SUBAPPLICATION Uebung_035a1_AX (* Ampelsteuerung mit Pattern Sequencer (AX) *)
  (* Standard: 61499-2; Description: Copyright (c) 2023 Meisterschulen am Ostbahnhof This program and the accompanying materials are made available under the terms of the Eclipse Public License 2.0 which is available at https://www.eclipse.org/legal/epl-2.0/ SPDX-License-Identifier: EPL-2.0 *)
  (* Version 1.0, 2026-02-01, Franz Höpfinger, Meisterschulen am Ostbahnhof, initial API and implementation and/or initial documentation *)
  PACKAGE Uebungen;
  IMPORT logiBUS::io::DI::logiBUS_DI::Input_I1;
  IMPORT logiBUS::io::DI::logiBUS_DI_Events::BUTTON_SINGLE_CLICK;
  IMPORT logiBUS::io::DQ::logiBUS_DO::Output_Q1;
  IMPORT logiBUS::io::DQ::logiBUS_DO::Output_Q2;
  IMPORT logiBUS::io::DQ::logiBUS_DO::Output_Q3;
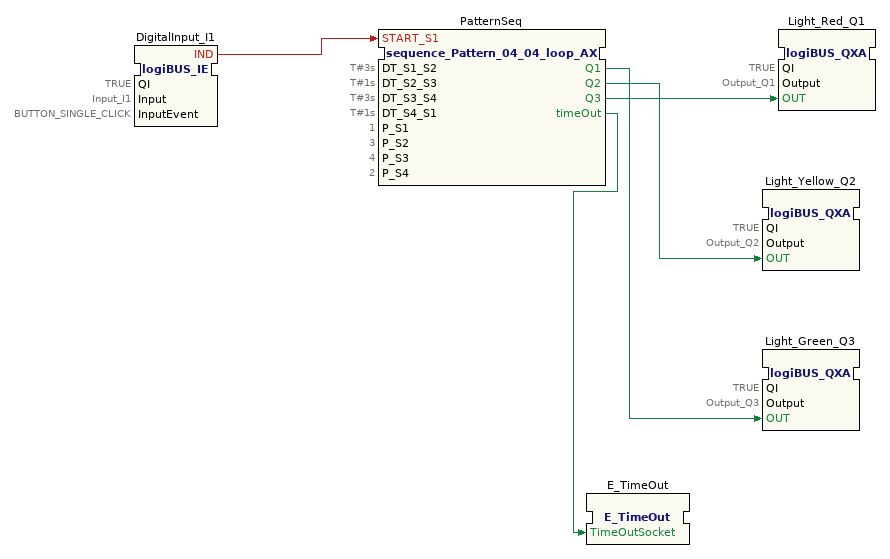
  FBS
    PatternSeq : logiBUS::utils::sequence::pattern::sequence_Pattern_04_04_loop_AX(DT_S1_S2 := T#3s, DT_S2_S3 := T#1s, DT_S3_S4 := T#3s, DT_S4_S1 := T#1s, P_S1 := 1, P_S2 := 3, P_S3 := 4, P_S4 := 2);
    DigitalInput_I1 : logiBUS::io::DI::logiBUS_IE(QI := TRUE, Input := Input_I1, InputEvent := BUTTON_SINGLE_CLICK);
    Light_Red_Q1 : logiBUS::io::DQ::logiBUS_QXA(QI := TRUE, Output := Output_Q1);
    Light_Yellow_Q2 : logiBUS::io::DQ::logiBUS_QXA(QI := TRUE, Output := Output_Q2);
    Light_Green_Q3 : logiBUS::io::DQ::logiBUS_QXA(QI := TRUE, Output := Output_Q3);
    E_TimeOut : iec61499::events::E_TimeOut;
  END_FBS
  EVENT_CONNECTIONS
    DigitalInput_I1.IND TO PatternSeq.START_S1;
  END_CONNECTIONS
  ADAPTER_CONNECTIONS
    PatternSeq.Q1 TO Light_Red_Q1.OUT;
    PatternSeq.Q2 TO Light_Yellow_Q2.OUT;
    PatternSeq.Q3 TO Light_Green_Q3.OUT;
    PatternSeq.timeOut TO E_TimeOut.TimeOutSocket;
  END_CONNECTIONS
END_SUBAPPLICATION
